// TIA Portal V16 export
// export: Created 2026-03-31T12:42:57.5562131Z, ExportSetting WithDefaults, DisplayName Totally Integrated Automation Portal, DisplayVersion V16, DisplayName TIA Portal Version Control Interface, DisplayVersion V16, DisplayName TIA Portal Openness, DisplayVersion V16, DisplayName STEP 7 Professional, DisplayVersion V16, DisplayName STEP 7 Safety, DisplayVersion V16, DisplayName WinCC Advanced, DisplayVersion V16
ORGANIZATION_BLOCK "OB82"   // OB82, FBD, DiagnosticErrorInterrupt
VERSION : 0.1
// stored: IsIECCheckEnabled false
   VAR_TEMP
      Temp_0 : Byte;
      Temp_1 : Byte;
      Temp_2 : Byte;
      Temp_3 : Byte;
      Temp_4 : Byte;
      Temp_5 : Byte;
      Temp_6 : Word;
      Temp_7 : Bool;
      Temp_8 : Bool;
      Temp_9 : Bool;
      Temp_10 : Bool;
      Temp_11 : Bool;
      Temp_12 : Bool;
      Temp_13 : Bool;
      Temp_14 : Bool;
      Temp_15 : Byte;
      Temp_16 : Bool;
      Temp_17 : Bool;
      Temp_18 : Bool;
      Temp_19 : Bool;
      Temp_20 : Bool;
      Temp_21 : Bool;
      Temp_22 : Bool;
      Temp_23 : Bool;
      Temp_24 : Bool;
      Temp_25 : Bool;
      Temp_26 : Bool;
      Temp_27 : Bool;
      Temp_28 : Bool;
      Temp_29 : Bool;
      Temp_30 : Bool;
      Temp_31 : Bool;
      Temp_32 : Date_And_Time;
   END_VAR
BEGIN
END_ORGANIZATION_BLOCK
